FUNCTION F_SINT_ARG : ST_Arg
VAR_INPUT
	nInput : SINT;
END_VAR
VAR
	stArg : ST_Arg;
	sysVar_Info : __SYSTEM.VAR_INFO;
END_VAR

sysVar_Info 	:= __VARINFO(nInput);
stArg.TypeClass := sysVar_Info.TypeClass;
stArg.pValue 	:= 0;
stArg.diSize 	:= SIZEOF(nInput);
stArg.sValue 	:= TO_STRING(nInput); 
F_SINT_ARG := stArg;

END_FUNCTION

(* stored: Version 1.1.0.1, ProductVersion 3.1.4024.4
   POU F_SINT_ARG: Id {5af99430-5c8f-4ead-bf48-b126248542da}, SpecialFunc None *)
